FUNCTION_BLOCK FB_StepManagerBasic_Test EXTENDS FB_TestSuite
VAR_INPUT
END_VAR
VAR_OUTPUT
END_VAR
VAR
END_VAR

RequestStep();
Reset();

METHOD RequestStep
VAR
	step_manager : StepManagerBasic();
END_VAR
TEST('RequestStep');
	step_manager._requestStep(2);
	AssertEquals_UDINT(Expected := 2, Actual := step_manager.currentStep, 'Current Step shall be requested step');
TEST_FINISHED();
END_METHOD

METHOD Reset
VAR
	step_manager : StepManagerBasic();
END_VAR
TEST('Reset');
	step_manager._requestStep(20);
	AssertEquals_UDINT(Expected := 20, Actual := step_manager.currentStep, 'Confirm current step is not default');
	
	step_manager._reset();
	AssertEquals_UDINT(Expected := SEQUENCE_STEP.NO_STEP, Actual := step_manager.currentStep, 'Reset should have put current step back to default');
TEST_FINISHED();
END_METHOD

END_FUNCTION_BLOCK

(* stored: Version 1.1.0.1
   POU FB_StepManagerBasic_Test: Id {f2f4fe9e-d358-482a-b327-02ec29657bd0}, SpecialFunc None
   Method RequestStep: Id {198c2120-5857-4c31-b6b8-c5eeca56d028}
   Method Reset: Id {f87175cc-f817-48db-aeb6-5cea267ae2ed} *)
